# EPICS substitutions: Db/seq-freia.substitutions
file "seq-freia-pmd-waveform.template" { pattern
{P,    ADC_CHAN}
{$(P), "0"}
{$(P), "1"}
{$(P), "2"}
{$(P), "3"}
{$(P), "4"}
{$(P), "5"}
{$(P), "6"}
{$(P), "7"}
{$(P), "8"}
{$(P), "9"}
{$(P), "10"}
{$(P), "11"}
{$(P), "12"}
{$(P), "13"}
{$(P), "14"}
{$(P), "15"}
}
